(* PLC project Sin nombre, Desconocido Sin nombre 1 *)
(* stored: creationDateTime 2021-11-16T16:25:21, modificationDateTime 2021-11-25T16:22:56 *)

PROGRAM program0
  VAR
    AtEmptyPallet AT %IX100.0 : BOOL := FALSE;
    AtLeftEntry AT %IX100.1 : BOOL := TRUE;
    AtLeftExit AT %IX100.2 : BOOL := TRUE;
    AtPopulatedPallet AT %IX100.3 : BOOL := FALSE;
    AtRightEntry AT %IX100.4 : BOOL := TRUE;
    AtRightExit AT %IX100.5 : BOOL := TRUE;
    AtSecondConveyorEntry AT %IX100.6 : BOOL := TRUE;
    EmptyPalletSensor AT %IX100.7 : BOOL := TRUE;
    FirstTransferLoaded AT %IX101.0 : BOOL := TRUE;
    HighSensor AT %IX101.1 : BOOL := TRUE;
    LowSensor AT %IX101.2 : BOOL := TRUE;
    PalletSensor AT %IX101.3 : BOOL := TRUE;
    PopulatedPalletSensor AT %IX101.4 : BOOL := TRUE;
    SecondTransferLoaded AT %IX101.5 : BOOL := TRUE;
    ThirdTransferLoaded AT %IX101.6 : BOOL := TRUE;
    ConveyorLeft AT %QX100.0 : BOOL := FALSE;
    ConveyorRight AT %QX100.1 : BOOL := FALSE;
    FirstConveyor AT %QX100.2 : BOOL := TRUE;
    LoadFirstTransfer AT %QX100.3 : BOOL := FALSE;
    LoadSecondTransfer AT %QX100.4 : BOOL := FALSE;
    LoadThirdTransfer AT %QX100.5 : BOOL := FALSE;
    RemoverEmptyPallet AT %QX100.6 : BOOL := FALSE;
    RemoverLargePackage AT %QX100.7 : BOOL := FALSE;
    RemoverSmallPackage AT %QX101.0 : BOOL := FALSE;
    SecondConveyor AT %QX101.1 : BOOL := FALSE;
    TransEmptyPallet AT %QX101.2 : BOOL := FALSE;
    TransPopulatedPallet AT %QX101.3 : BOOL := FALSE;
    TransToSecondConveyor AT %QX101.4 : BOOL := FALSE;
    TransfLeft AT %QX101.5 : BOOL := FALSE;
    TransfRight AT %QX101.6 : BOOL := FALSE;
  END_VAR
  VAR
    PopulatedPallet : RS;
    TOF0 : TOF;
    TOF1 : TOF;
    High : RS;
    TOF2 : TOF;
    TOF3 : TOF;
    RS0 : RS;
  END_VAR
  VAR  (* added by the conversion: wires and edge detectors of the diagram *)
    _AND74_OUT : BOOL;
    _NOT2_OUT : BOOL;
  END_VAR

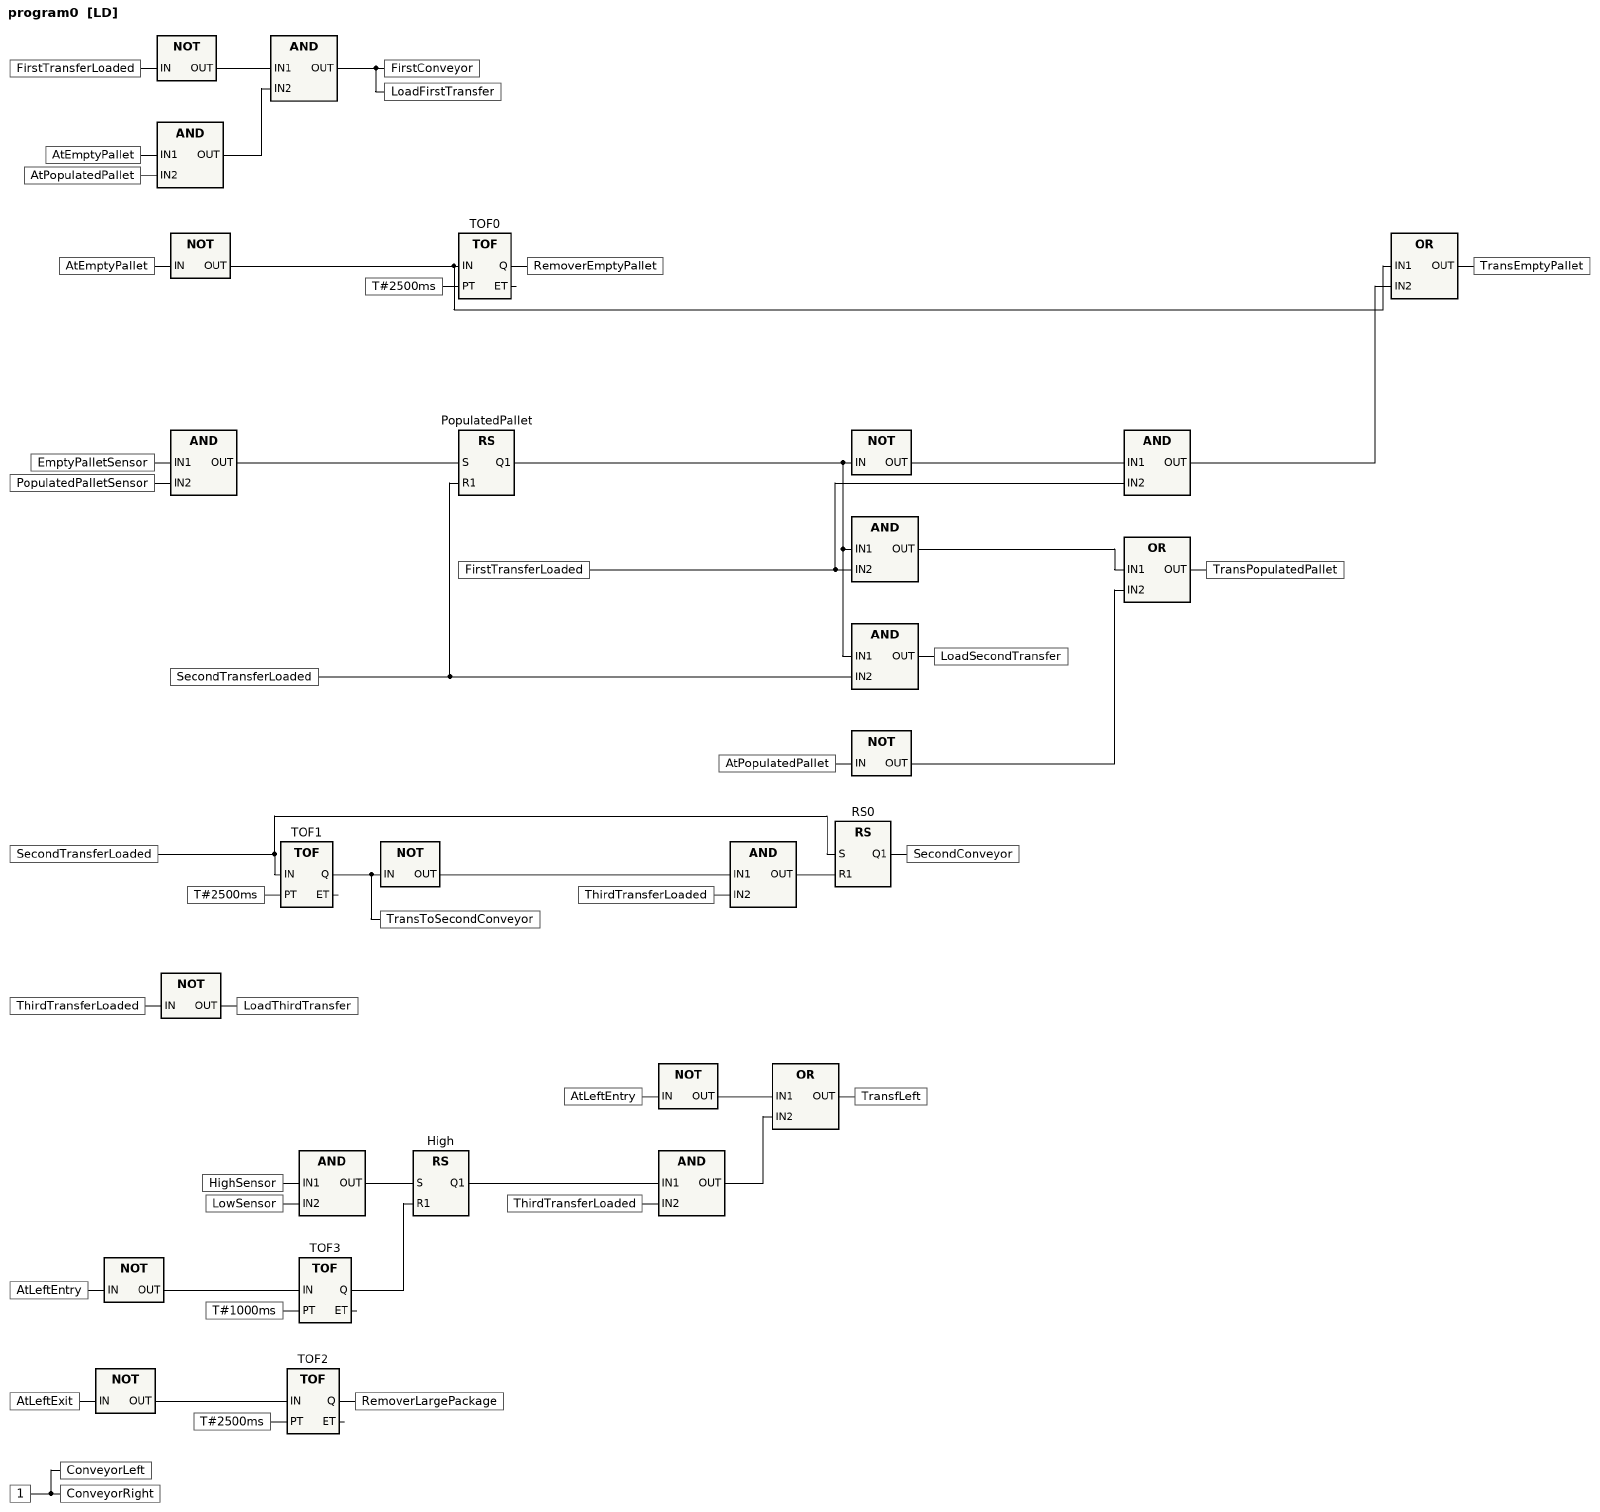
(* LD diagram, written out as Structured Text *)
_AND74_OUT := NOT FirstTransferLoaded AND AtEmptyPallet AND AtPopulatedPallet;
FirstConveyor := _AND74_OUT;
LoadFirstTransfer := _AND74_OUT;
_NOT2_OUT := NOT AtEmptyPallet;
TOF0(IN := _NOT2_OUT, PT := T#2500ms);
RemoverEmptyPallet := TOF0.Q;
PopulatedPallet(S := EmptyPalletSensor AND PopulatedPalletSensor, R1 := SecondTransferLoaded);
TransEmptyPallet := _NOT2_OUT OR NOT PopulatedPallet.Q1 AND FirstTransferLoaded;
LoadSecondTransfer := PopulatedPallet.Q1 AND SecondTransferLoaded;
TransPopulatedPallet := PopulatedPallet.Q1 AND FirstTransferLoaded OR NOT AtPopulatedPallet;
TOF1(IN := SecondTransferLoaded, PT := T#2500ms);
TransToSecondConveyor := TOF1.Q;
RS0(S := SecondTransferLoaded, R1 := NOT TOF1.Q AND ThirdTransferLoaded);
SecondConveyor := RS0.Q1;
LoadThirdTransfer := NOT ThirdTransferLoaded;
TOF3(IN := NOT AtLeftEntry, PT := T#1000ms);
High(S := HighSensor AND LowSensor, R1 := TOF3.Q);
TransfLeft := NOT AtLeftEntry OR High.Q1 AND ThirdTransferLoaded;
ConveyorLeft := 1;
ConveyorRight := 1;
TOF2(IN := NOT AtLeftExit, PT := T#2500ms);
RemoverLargePackage := TOF2.Q;
END_PROGRAM

CONFIGURATION Config0
  RESOURCE Res0 ON PLC
    TASK task0(INTERVAL := T#20ms, PRIORITY := 0);
    PROGRAM instance0 WITH task0 : program0;
  END_RESOURCE
END_CONFIGURATION
